INTERFACE I_ManualImplementation_1

PROPERTY ipManualControl : Array [0..10, 0..10] of I_ManualControl
GET
END_GET
END_PROPERTY

END_INTERFACE

(* stored: Version 1.1.0.1, ProductVersion 3.1.4024.5
   Itf I_ManualImplementation_1: Id {c88c4bf4-402e-4185-90df-d2ecc5fa3db8}
   Property ipManualControl: Id {a7e1bbad-d3e1-4dd3-b266-295d3d5931bf}
   Get Get: Id {be53d314-55a1-41f9-bc85-9bb46f75cea5} *)
